(* IEC 61131-3 sources: Industry-PLC-LLM/data/PLCBEAD_repo/PLCBEAD_PLCEmbed-main/PLC-BEAD/Source/GEB/SCALE_B4, 1 file *)

(* ---- SCALE_B4.ST ---- *)
FUNCTION _BYTE_TO_REAL:REAL
	VAR_INPUT
		IN :	BYTE;
	END_VAR

	_BYTE_TO_REAL := USINT_TO_REAL(BYTE_TO_USINT(IN));
END_FUNCTION

FUNCTION SCALE_B4:REAL

	VAR_INPUT
		IN1 :	BYTE;
		IN2 :	BYTE;
		IN3 :	BYTE;
		IN4 :	BYTE;
		K :	REAL;
		O :	REAL;
		IN1_MIN :	REAL;
		IN1_MAX :	REAL;
		IN2_MIN :	REAL;
		IN2_MAX :	REAL;
		IN3_MIN :	REAL;
		IN3_MAX :	REAL;
		IN4_MIN :	REAL;
		IN4_MAX :	REAL;
	END_VAR

	SCALE_B4 := 	(((IN1_max - IN1_min)* _BYTE_TO_REAL(IN1) + (IN2_max - IN2_min)* _BYTE_TO_REAL(IN2) + (IN3_max - IN3_min)* _BYTE_TO_REAL(IN3) + (in4_max - in4_min)* _BYTE_TO_REAL(in4))* 0.003921569 + IN1_mIN + IN2_mIN + IN3_mIN + in4_min) * K + O;

END_FUNCTION

PROGRAM program0
  VAR
	IN1 :	BYTE;
	IN2 :	BYTE;
	IN3 :	BYTE;
	IN4 :	BYTE;
	K :	REAL;
	O :	REAL;
	IN1_MIN :	REAL;
	IN1_MAX :	REAL;
	IN2_MIN :	REAL;
	IN2_MAX :	REAL;
	IN3_MIN :	REAL;
	IN3_MAX :	REAL;
	IN4_MIN :	REAL;
	IN4_MAX :	REAL;
	CEIL5_OUT : REAL;
  END_VAR

  CEIL5_OUT := SCALE_B4(IN1, IN2, IN3, IN4, K, O, IN1_MIN, IN1_MAX, IN2_MIN, IN2_MAX, IN3_MIN, IN3_MAX, IN4_MIN, IN4_MAX);

END_PROGRAM
